FUNCTION_BLOCK FB_Test
VAR_INPUT
	bVentil : BOOL;
	
END_VAR
VAR_OUTPUT
	bDoorC : BOOL;
	bDoorO : BOOL;
END_VAR
VAR
	nCounter : INT := 0;
	timer : TON;
END_VAR

IF bVentil THEN
	bDoorC := FALSE;
	timer(IN:= NOT bDoorC , PT:= T#5S , Q=> bDoorO := TRUE , ET=> );
	//bDoorO := TRUE;
	
END_IF

IF NOT bVentil THEN
	bDoorO := FALSE;
	timer(IN:= NOT bDoorO , PT:= T#5S , Q=> bDoorC := TRUE , ET=> );
	//bDoorC := TRUE;
END_IF

//Funktioniert nicht !

END_FUNCTION_BLOCK

(* stored: Version 1.1.0.1, ProductVersion 3.1.4024.15
   POU FB_Test: Id {d548480f-9773-47f3-b7ee-df6e2946a893}, SpecialFunc None *)
